(* CODESYS project system_lib.library
   Author: prg
   Version: 3.5.10.40
   Description: cystem lib for system command
   Title: cyber system lib
   Company: cyber

Project tree, tasks and I/O mapping:
  function do_system [ST]
*)

// do_system
FUNCTION do_system : INT
VAR_INPUT
	cmd : STRING(255);
END_VAR
VAR
END_VAR

END_FUNCTION
